RoboDK station: ABB.rdk

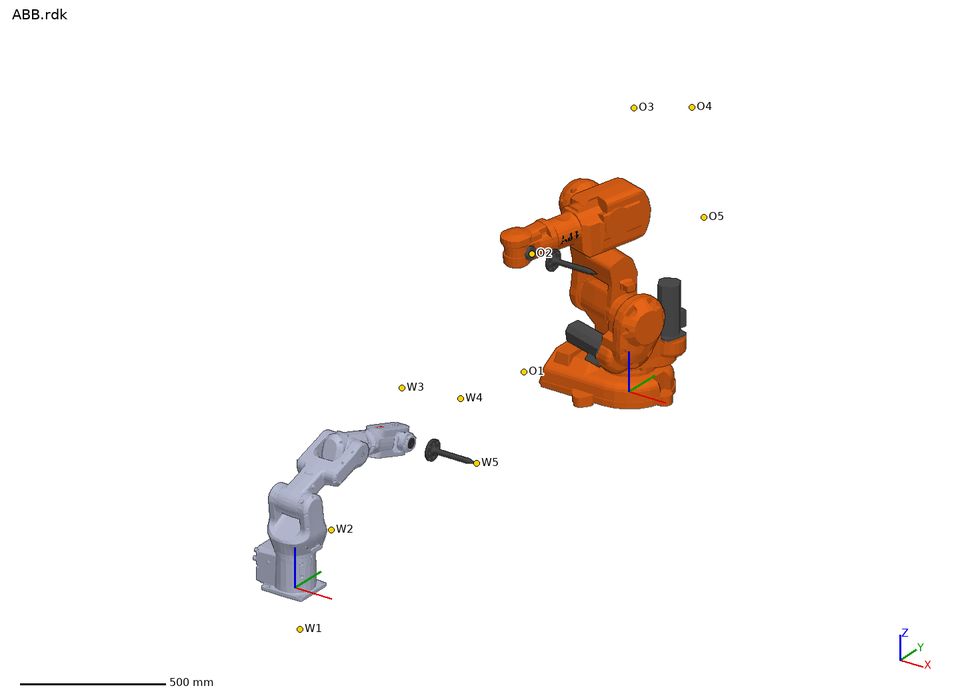
[picture v0: the station drawn from its stored meshes, robots at their saved joint values, targets as dots, program paths as lines]
Station ABB (saved by RoboDK 5.6.7). Poses are relative to the parent item; angles as X-Y-Z fixed-axis rotations.
Station parameters (name, value as stored): LIN64
  - frame ABB IRB 1100-4/0.58 Base at (0, 0, 0) mm
    - robot ABB IRB 1100-4/0.58: 6 axes, payload 4 kg, reach 580 mm, repeatability 0.01 mm, weight 21 kg
        modified DH rows (alpha deg, a mm, theta deg, d mm): 0, 0, 0, 327; -90, 0, -90, 0; 0, 280, 0, 0; -90, 10, 0, 300; 90, 0, 0, 0; -90, 0, 180, 64
        joint limits [-230, -115, -205, -230, -125, -400] to [230, 113, 55, 230, 125, 400]; home [0, 0, 0, 0, 0, 0]; saved at [85.862, 67.159, -50.998, -91.154, 86.025, 106.2]
      - tool Pointer, TCP at (0, 0, 274) mm, size 79 x 79 x 190 mm
    - target W1 (Cartesian target) at (364, -492.81, 139.22) mm, rotated rx 0 ry 90 rz 0 deg; joints [-86.98, 85.43, -39.102, -87.815, -87.915, 43.632] of ABB IRB 1100-4/0.58
    - target W2 (Cartesian target) at (377.62, -323.9, 456.71) mm, rotated rx 0 ry 90 rz 0 deg; joints [-83.027, 12.902, 17.505, -86.457, -83.99, 59.407] of ABB IRB 1100-4/0.58
    - target W3 (Cartesian target) at (377.62, 100.48, 829.21) mm, rotated rx 0 ry 90 rz 0 deg; joints [68.481, -16.624, -32.66, -73.361, 76.156, 38.682] of ABB IRB 1100-4/0.58
    - target W4 (Cartesian target) at (377.62, 451.55, 648.64) mm, rotated rx 0 ry 90 rz 0 deg; joints [84.986, 37.37, -54.742, -88.499, 85.215, 72.566] of ABB IRB 1100-4/0.58
    - target W5 (Cartesian target) at (377.62, 547.54, 361.8) mm, rotated rx 0 ry 90 rz 0 deg; joints [85.862, 67.159, -50.998, -91.154, 86.025, 106.2] of ABB IRB 1100-4/0.58
  - frame ABB IRB 140-6/0.8 Base at (0, 2000, -50) mm
    - robot ABB IRB 140-6/0.8: 6 axes, payload 6 kg, reach 810 mm, repeatability 0.03 mm, weight 98 kg
        modified DH rows (alpha deg, a mm, theta deg, d mm): 0, 0, 0, 352; -90, 70, -90, 0; 0, 360, 0, 0; -90, 0, 0, 380; 90, 0, 0, 0; -90, 0, 180, 65
        joint limits [-180, -90, -230, -200, -120, -400] to [180, 110, 50, 200, 120, 400]; home [0, 0, 0, 0, 0, 0]; saved at [-107.477, 6.159, -3.253, -90.914, -107.454, 86.954]
      - tool Pointer, TCP at (0, 0, 274) mm, size 79 x 79 x 190 mm
    - target O1 (Cartesian target) at (17.41, -655.53, 341.31) mm, rotated rx 0 ry 90 rz 0 deg; joints [-94.152, 52.374, -15.036, -92.521, -93.3, 52.59] of ABB IRB 140-6/0.8
    - target O2 (Cartesian target) at (-81.6, -465.6, 690.66) mm, rotated rx 0 ry 90 rz 0 deg; joints [-107.477, 6.159, -3.253, -90.914, -107.454, 86.954] of ABB IRB 140-6/0.8
    - target O3 (Cartesian target) at (-81.6, 145.77, 1003.05) mm, rotated rx 0 ry 90 rz 0 deg; joints [135.162, 38.601, -141.97, -134.375, 80.564, -9.513] of ABB IRB 140-6/0.8
    - target O4 (Cartesian target) at (-81.6, 492.16, 867.7) mm, rotated rx 0 ry 90 rz 0 deg; joints [106.587, 16.832, -43.596, 82.36, -104.767, 242.244] of ABB IRB 140-6/0.8
    - target O5 (Cartesian target) at (-81.6, 563.31, 417.71) mm, rotated rx 0 ry 90 rz 0 deg; joints [104.588, 35.315, 1.564, 98.877, -101.623, 307.784] of ABB IRB 140-6/0.8
  - Python program move (listed below)

--- Python program move ---
import cv2 as cv
import mediapipe as mp
from robodk import robolink    # RoboDK API

RDK = robolink.Robolink()

white = RDK.Item('ABB IRB 1100-4/0.58')
orange = RDK.Item('ABB IRB 140-6/0.8')
target1l = RDK.Item('W1')
target2l = RDK.Item('W2')
target3l = RDK.Item('W3')
target4l = RDK.Item('W4')
target5l = RDK.Item('W5')
target1r = RDK.Item('O1')
target2r = RDK.Item('O2')
target3r = RDK.Item('O3')
target4r = RDK.Item('O4')
target5r = RDK.Item('O5')

finger_tips = [8, 12, 16, 20]
vid = cv.VideoCapture(0)
mp_hands = mp.solutions.hands
mp_draw = mp.solutions.drawing_utils
hands = mp_hands.Hands()

def recognize_hands(x_coord, y_coord):
	num_arr = []
	if abs(x_coord[13]-x_coord[4]) > 50:
		num_arr.append(1)
	else:
		num_arr.append(0)
	for f in finger_tips:
		if y_coord[f] < y_coord[f-2]:
			num_arr.append(1)
		else:
			num_arr.append(0)
	return num_arr

while True:
	_, img = vid.read()
	img = cv.flip(img, 1)
	h, w, d = img.shape
	result = hands.process(cv.cvtColor(img, cv.COLOR_BGR2RGB))

	if result.multi_hand_landmarks:
		rx_coord = []
		ry_coord = []
		lx_coord = []
		ly_coord = []

		if len(result.multi_hand_landmarks) == 1:
			landmarks = result.multi_hand_landmarks[0]
			if (result.multi_handedness[0].classification[0].label == 'Right') and (result.multi_handedness[0].classification[0].score > 0.95):
				for l in landmarks.landmark:
					x = int(w*l.x)
					y = int(h*l.y)

					rx_coord.append(x)
					ry_coord.append(y)

			elif (result.multi_handedness[0].classification[0].label == 'Left') and (result.multi_handedness[0].classification[0].score > 0.95):
				for l in landmarks.landmark:
					x = int(w*l.x)
					y = int(h*l.y)

					lx_coord.append(x)
					ly_coord.append(y)

			else:
				continue

			mp_draw.draw_landmarks(img, landmarks, mp_hands.HAND_CONNECTIONS)

		elif len(result.multi_hand_landmarks) == 2:
			if (result.multi_handedness[0].classification[0].label == 'Left' and result.multi_handedness[0].classification[0].score > 0.95) or (result .multi_handedness[1].classification[0].label == 'Right' and result.multi_handedness[1].classification[0].score > 0.95):
				left_landmarks = result.multi_hand_landmarks[0]
				right_landmarks = result.multi_hand_landmarks[1]
			elif (result.multi_handedness[0].classification[0].label == 'Right' and result.multi_handedness[0].classification[0].score > 0.95) or (result .multi_handedness[1].classification[0].label == 'Left' and result.multi_handedness[1].classification[0].score > 0.95):
				left_landmarks = result.multi_hand_landmarks[1]
				right_landmarks = result.multi_hand_landmarks[0]
			else:
				continue

			for l in right_landmarks.landmark:
				x = int(w*l.x)
				y = int(h*l.y)

				rx_coord.append(x)
				ry_coord.append(y)

			for l in left_landmarks.landmark:
				x = int(w*l.x)
				y = int(h*l.y)

				lx_coord.append(x)
				ly_coord.append(y)

			mp_draw.draw_landmarks(img, right_landmarks, mp_hands.HAND_CONNECTIONS)
			mp_draw.draw_landmarks(img, left_landmarks, mp_hands.HAND_CONNECTIONS)

		if len(lx_coord) != 0:
			left_finger_arr = recognize_hands(lx_coord, ly_coord)

			if left_finger_arr == [0,1,0,0,0]:
				cv.putText(img, 'Left: 1', (50,100), cv.FONT_HERSHEY_COMPLEX, 1, (255,0,0), thickness=1)
				white.MoveJ(target1l)
				white.RunInstruction('Program_Done')

			if left_finger_arr == [0,1,1,0,0]:
				cv.putText(img, 'Left: 2', (50,100), cv.FONT_HERSHEY_COMPLEX, 1, (255,0,0), thickness=1)
				white.MoveJ(target2l)
				white.RunInstruction('Program_Done')

			if left_finger_arr == [0,1,1,1,0]:
				cv.putText(img, 'Left: 3', (50,100), cv.FONT_HERSHEY_COMPLEX, 1, (255,0,0), thickness=1)
				white.MoveJ(target3l)
				white.RunInstruction('Program_Done')

			if left_finger_arr == [0,1,1,1,1]:
				cv.putText(img, 'Left: 4', (50,100), cv.FONT_HERSHEY_COMPLEX, 1, (255,0,0), thickness=1)
				white.MoveJ(target4l)
				white.RunInstruction('Program_Done')

			if left_finger_arr == [1,1,1,1,1]:
				cv.putText(img, 'Left: 5', (50,100), cv.FONT_HERSHEY_COMPLEX, 1, (255,0,0), thickness=1)
				white.MoveJ(target5l)
				white.RunInstruction('Program_Done')

		if len(rx_coord) != 0:
			right_finger_arr = recognize_hands(rx_coord, ry_coord)

			if right_finger_arr == [0,1,0,0,0]:
				cv.putText(img, 'Right: 1', (450,100), cv.FONT_HERSHEY_COMPLEX, 1, (0,0,255), thickness=1)
				orange.MoveJ(target1r)
				orange.RunInstruction('Program_Done')

			if right_finger_arr == [0,1,1,0,0]:
				cv.putText(img, 'Right: 2', (450,100), cv.FONT_HERSHEY_COMPLEX, 1, (0,0,255), thickness=1)
				orange.MoveJ(target2r)
				orange.RunInstruction('Program_Done')

			if right_finger_arr == [0,1,1,1,0]:
				cv.putText(img, 'Right: 3', (450,100), cv.FONT_HERSHEY_COMPLEX, 1, (0,0,255), thickness=1)
				orange.MoveJ(target3r)
				orange.RunInstruction('Program_Done')

			if right_finger_arr == [0,1,1,1,1]:
				cv.putText(img, 'Right: 4', (450,100), cv.FONT_HERSHEY_COMPLEX, 1, (0,0,255), thickness=1)
				orange.MoveJ(target4r)
				orange.RunInstruction('Program_Done')

			if right_finger_arr == [1,1,1,1,1]:
				cv.putText(img, 'Right: 5', (450,100), cv.FONT_HERSHEY_COMPLEX, 1, (0,0,255), thickness=1)
				orange.MoveJ(target5r)
				orange.RunInstruction('Program_Done')

	cv.imshow('Vid',img)
	cv.waitKey(1)
